{region '#Template'}
	{attribute 'Version' := '5.0.0.0'}
	{attribute 'Tags' := '"LCID": "1031", "Text": "Fassade, Sonnenschutz, Dämmerungsautomatik"'}
	{attribute 'Tags' := '"LCID": "1033", "Text": "Facade, Sunprotection, twilight-automatic"'}
	{attribute 'Using' := '"Type": "Template", "URI": "ST_BA_SunBld"'}
	{attribute 'Using' := '"Type": "Template", "URI": "E_BA_SunBldPrio"'}
	{attribute 'Description' := '"LCID": "1031", "Text": "Sonnenschutz fassadenweise Dämmerungsautomatik"'}
	{attribute 'Description' := '"LCID": "1033", "Text": "Sunprotection facade-twilightautomatic"'}
{endregion}
FUNCTION_BLOCK FB_BA_Facade_TwilightAutomatic EXTENDS FB_BA_View
VAR_INPUT
END_VAR
VAR_OUTPUT
	stSunBld					: ST_BA_SunBld;
	bTwiLgtAutoEvent			: BOOL;	
END_VAR
VAR_INPUT CONSTANT
	FcdTwiLgtAutoEn				: FB_BA_BV_Op;		
	FcdTwiLgtAutoEvent			: FB_BA_SunBldEvt :=(ePrio:=E_BA_SunBldPrio.eFacadeTwilightAutomatic);		
END_VAR
VAR
END_VAR

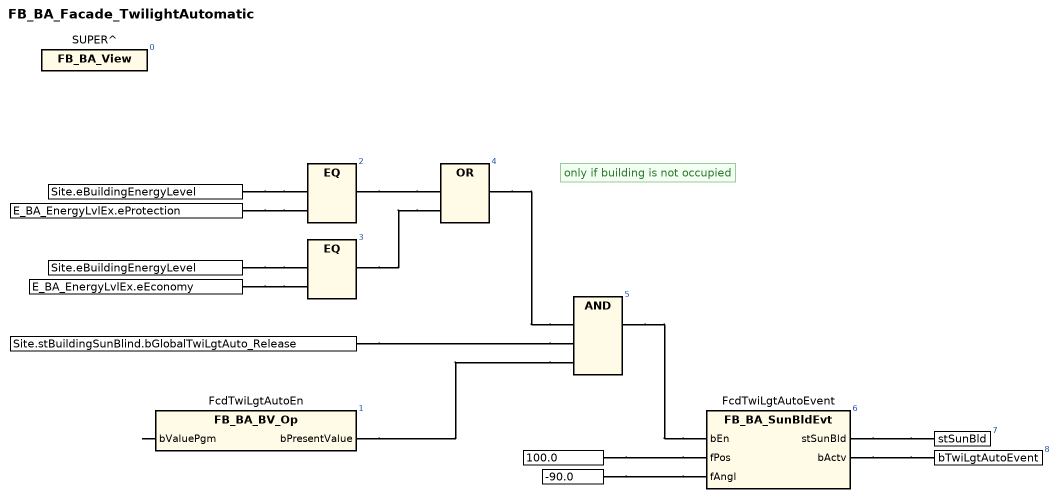
SUPER^(); // FB_BA_View
FcdTwiLgtAutoEn(); // FB_BA_BV_Op
// only if building is not occupied
FcdTwiLgtAutoEvent(
    bEn := (Site.eBuildingEnergyLevel = E_BA_EnergyLvlEx.eProtection OR Site.eBuildingEnergyLevel = E_BA_EnergyLvlEx.eEconomy) AND Site.stBuildingSunBlind.bGlobalTwiLgtAuto_Release AND FcdTwiLgtAutoEn.bPresentValue,
    fPos := 100.0,
    fAngl := -90.0); // FB_BA_SunBldEvt
stSunBld := FcdTwiLgtAutoEvent.stSunBld;
bTwiLgtAutoEvent := FcdTwiLgtAutoEvent.bActv;

METHOD FB_init : BOOL
VAR_INPUT
	bInitRetains : BOOL; // if TRUE; the retain variables are initialized (warm start / cold start)
	bInCopyCode : BOOL;  // if TRUE; the instance afterwards gets moved into the copy code (online change)
END_VAR
FcdTwiLgtAutoEn.iParent			:= THIS^;
FcdTwiLgtAutoEn.iLabel			:= LblCtl_FacadeTwilightAutomaticEnable;	
FcdTwiLgtAutoEn.sObjectName		:= '{Idx=01}';
FcdTwiLgtAutoEn.sInactiveText	:= txtEvent_Off;
FcdTwiLgtAutoEn.sActiveText		:= txtEvent_On;
FcdTwiLgtAutoEn.bValueRm		:= FALSE;
FcdTwiLgtAutoEn.eToggleMode		:= E_BA_ToggleMode.eSwitch;
END_METHOD

END_FUNCTION_BLOCK

(* stored: Version 1.1.0.1, ProductVersion 3.1.4024.12
   POU FB_BA_Facade_TwilightAutomatic: Id {0934b42c-703e-4c56-83de-ae24e98dd0b1}, SpecialFunc None
   Method FB_init: Id {006204e6-a758-46b5-bf94-07fad241d64e} *)
